{attribute 'GeneratedUsingTerminal: EL3314-0000-0016'}
{attribute addProperty BoxType "EL3314-0000-0016"}
{attribute addProperty Id "EtcSlaveTerminalBaseTC_Inputs_Channel_1AT %I*TC_Inputs_Channel_EA9DF21E9TC_Inputs_Channel_2AT %I*TC_Inputs_Channel_EA9DF21E9TC_Inputs_Channel_3AT %I*TC_Inputs_Channel_EA9DF21E9TC_Inputs_Channel_4AT %I*TC_Inputs_Channel_EA9DF21E9WcStateAT %I*WcState_9091E0EB2InfoDataAT %I*InfoData_32EB74EA10"}
{attribute addProperty CRC "3307028514"}
{attribute addProperty Size "48"}
TYPE EL3314_C51D4022 EXTENDS EtcSlaveTerminalBase :
STRUCT
	{attribute addProperty Name "TC_Inputs_Channel_1"}
	TC_Inputs_Channel_1 : TC_Inputs_Channel_EA9DF21E;
	{attribute addProperty Name "TC_Inputs_Channel_2"}
	TC_Inputs_Channel_2 : TC_Inputs_Channel_EA9DF21E;
	{attribute addProperty Name "TC_Inputs_Channel_3"}
	TC_Inputs_Channel_3 : TC_Inputs_Channel_EA9DF21E;
	{attribute addProperty Name "TC_Inputs_Channel_4"}
	TC_Inputs_Channel_4 : TC_Inputs_Channel_EA9DF21E;
	{attribute addProperty Name "WcState"}
	WcState : WcState_9091E0EB;
	{attribute addProperty Name "InfoData"}
	InfoData : InfoData_32EB74EA;
END_STRUCT
END_TYPE

(* stored: Version 1.2.0.0, ProductVersion 3.1.4024.9
   DUT EL3314_C51D4022: Id {508ef5d2-a2f6-48ec-926d-812fe95ead2f} *)
